(* Logix 5000 project; controller DispersionPlc vendor 1 type 14 code 108 rev 34.11; software revision 34.01; part 4 of 22 *)
(* tags used below, declared in another part *)
   _JISdebug : DINT;
   AFI : BOOL;
   B4320_HighHighLevel : BOOL;
   B4320_HighLevel : BOOL;
   B4320_OkToRun : BOOL;
   B4320_PumpAutoCommand : BOOL;
   B4320_Selected : BOOL;
   B4320_SelectPB : BOOL;
   B4320_Toggle : AOI_Toggle;
   B4320_Transfer : BOOL;
   B4320_transfer_amount : REAL;
   B4320_TransferLimit : REAL;
   B4320_transferLimitMessage : BOOL;
   B4320_TransferSetpoint : REAL;
   B4320_TransferStarted : BOOL;
   B4320_TransferStartPB : BOOL;
   B4320_TransferStopPB : BOOL;
   BL_4310_AUX : ALIAS FOR Local:1:I.Data[1].2;
   BL_4310_RUN : ALIAS FOR Local:1:O.Data[0].2;
   BLANK64 : Stp64;
   bogus_bit : BOOL;
   Cat_Pump_manual : BOOL;
   Cat_Recirc_Transfer_T430X : Seq64;
   Cat_Scale_Factor : REAL;
   cat_start_dispencse : BOOL;
   Cat_Tank_Destination : DINT;
   cat_target_weight_bypass : BOOL;
   Cat_Zero : REAL;
   catalyst_MaxFeedRate : REAL;
   CATALYST_RESET : BOOL;
   CatalystTimers_11_HMI : REAL;
   CE_4301 : REAL;
   CE_4301_OffSet : REAL;
   CE_4301_Sf : REAL;
   CurrentTrasferredLb : REAL;
   dan5 : BOOL;
   DATAFDUNLATCH : TIMER;
   DATAUNCOUNT : COUNTER;
   DispersionAlarms : BOOL[256];
   DPT_4301 : REAL;
   DPT_4301_Holding : REAL;
   DPT_4301_OffSet : REAL;
   DPT_4301_Samples : DINT;
   DPT_4301_Sf : REAL;
   DPT_4302 : REAL;
   DPT_4302_Holding : REAL;
   DPT_4302_OffSet : REAL;
   DPT_4302_Samples : DINT;
   DPT_4302_Sf : REAL;
   DPT_4303 : REAL;
   DPT_4303_Holding : REAL;
   DPT_4303_OffSet : REAL;
   DPT_4303_Samples : DINT;
   DPT_4303_Sf : REAL;
   DPT_4320 : REAL;
   Emergency_Cool_4301 : BOOL;
   Estop_Disp : ALIAS FOR Local:3:I.Data.1;
   Estop_Inx : ALIAS FOR Local:3:I.Data.3;
   FE_4303 : REAL;
   FE_4303_AOI : Analog_Scale;
   FE_4303_Corrected : REAL;
   FE_4303_Correction_Sf : REAL;
   FE_4303_OffSet : REAL;
   FE_4303_OffSet_Out : REAL;
   FE_4303_Out : REAL;
   FE_4304 : REAL;
   FE_4304_AOI : Analog_Scale;
   FE_4304_OffSet : REAL;
   FE_4304_Sf : REAL;
   FE_4305 : REAL;
   FE_4305_OffSet : REAL;
   FE_4305_Sf : REAL;
   INX_Alarm : BOOL[32];
   INX_AlarmTmr : TIMER[32];
   InxAlarms : BOOL[128];
   LS_4302_Raw : INT;
   MAINT_SV4304_02_PB : BOOL;
   MAINT_SV4304_03_PB : BOOL;
   MAINT_XV4304_04_PB : BOOL;
   MIXER_A_4304_RUN : ALIAS FOR Local:1:O.Data[0].16;
   MMI_A_4304_RUN_PB : BOOL;
   MMI_B4320_Level : INT;
   MMI_Cat_Nit_Purge_Time : REAL;
   MMI_Cat_Recirc_Pump_Speed : REAL;
   MMI_P_4304_RUN_PB : BOOL;
   MMI_P_4320_RUN_PB : BOOL;
   MMI_SV4304_02_PB : BOOL;
   MMI_SV4304_03_PB : BOOL;
   MMI_SV4304_PB : BOOL;
   MMI_T4301_Level : INT;
   MMI_T4302_Level : INT;
   MMI_V4304_Acc_Weight : REAL;
   MMI_V4304_Acc_Weight_Temp : REAL;
   MMI_V4304_TransTime_SP : REAL;
   MMI_V4304_Weight_SP : REAL;
   MMI_W4303_Level : INT;
   MMI_XV4304_02_PB : BOOL;
   MMI_XV4304_03_PB : BOOL;
   MMI_XV4304_04_PB : BOOL;
   MMI_XV_4304_01_PB : BOOL;
   O5_6_PL : ALIAS FOR Local:5:O.Data.14;
   O5_9_PL : ALIAS FOR Local:5:O.Data.9;
   O7_11_BEC : ALIAS FOR Local:7:O.Data.11;
   ONS101 : BOOL;
   PLCStatus : AStd_PLCStatus;
   S47_HighHighLevel : BOOL;
   S47_SelectPB : BOOL;
   S47_TransferStarted : BOOL;
   SPARE_O603 : ALIAS FOR Local:6:O.Data.3;
   SPARE_O604 : ALIAS FOR Local:6:O.Data.4;
   SRT_PB_BL_4310 : ALIAS FOR Local:2:I.Data.13;
   SRT_PB_P_4310 : ALIAS FOR Local:2:I.Data.15;
   STP_PB_BL_4310 : ALIAS FOR Local:2:I.Data.14;
   STP_PB_P_4310 : ALIAS FOR Local:3:I.Data.0;
   SV_4304 : ALIAS FOR Local:5:O.Data.11;
   SV_4304_02 : BOOL;
   SV_4304_02_Enable_PB : BOOL;
   SV_4304_03 : BOOL;
   SV_4304_03_Enable_PB : BOOL;
   SV_4310 : ALIAS FOR Local:5:O.Data.5;
   T4301_AIR_PURGE_AUTO : BOOL;
   T4301_AIR_PURGE_REQUEST : BOOL;
   T4301_COOLING_NOT_PURGED : BOOL;
   T4301_COOLING_OCCURED : BOOL;
   T4301_COOLING_OPERATION : BOOL;
   T4301_K : Kettle;
   T4301_Manual_AIR_PURGE_REQUEST : BOOL;
   T4301_Mixer : VFD;
   T4301_Post_PurgeTm : DINT;
   T4301_Pre_PurgeTm : DINT;
   T4301_Process_Alarm_Setpoints : Alarm_SPT;
   T4301_Purge_Complete : BOOL;
   T4301_Request_Cooling_Tmr : TIMER[5];
   T4301Purge : Seq64;
   T_4301_Temp_Holding : REAL;
   T_4301_Temp_Samples : REAL;
   Task_Permissive : DINT[2];
   TE_4301A : ALIAS FOR Local:8:I.Ch0Data;
   TOGGLE : BOOL;
   TransferDone : BOOL;
   TransferSetpoint : REAL;
   V4304_Pump : VFD;
   V4304_Pump_TargetDriveSpeed_Timer : TIMER;
   XV_4304 : ALIAS FOR Local:5:O.Data.4;
   XV_4304_02 : BOOL;
   XV_4304_03 : BOOL;
   XV_4304_04 : BOOL;
   XV_S47_1_CloseCommand : BOOL;
   XV_S47_1_IsClosed : BOOL;
   XV_S47_1_IsOpen : BOOL;
   XV_S47_1_OpenCommand : BOOL;
   XV_S47_2_CloseCommand : BOOL;
   XV_S47_2_IsClosed : BOOL;
   ZSO_4304_02 : BOOL;
   ZSO_4304_03 : BOOL;
(* General_Purpose, continued *)

ROUTINE TimeSync   (* ladder *)
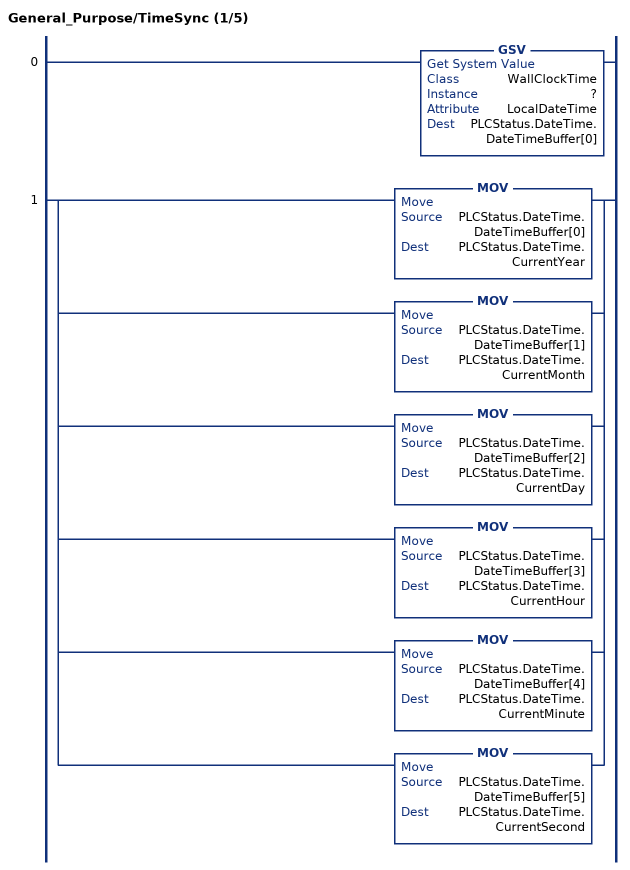
   0: GSV(WallClockTime,?,LocalDateTime,PLCStatus.DateTime.DateTimeBuffer[0]);
   1: [MOV(PLCStatus.DateTime.DateTimeBuffer[0],PLCStatus.DateTime.CurrentYear) ,MOV(PLCStatus.DateTime.DateTimeBuffer[1],PLCStatus.DateTime.CurrentMonth) ,MOV(PLCStatus.DateTime.DateTimeBuffer[2],PLCStatus.DateTime.CurrentDay) ,MOV(PLCStatus.DateTime.DateTimeBuffer[3],PLCStatus.DateTime.CurrentHour) ,MOV(PLCStatus.DateTime.DateTimeBuffer[4],PLCStatus.DateTime.CurrentMinute) ,MOV(PLCStatus.DateTime.DateTimeBuffer[5],PLCStatus.DateTime.CurrentSecond) ];
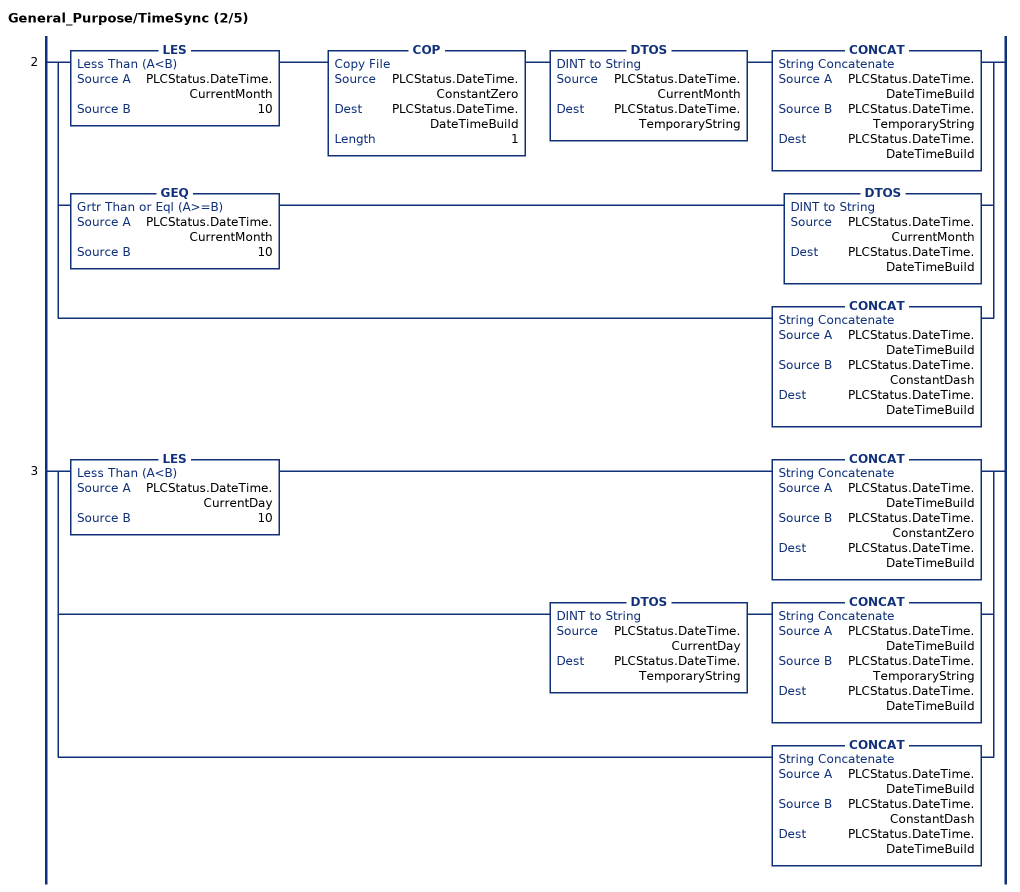
   2: [LES(PLCStatus.DateTime.CurrentMonth,10) COP(PLCStatus.DateTime.ConstantZero,PLCStatus.DateTime.DateTimeBuild,1) DTOS(PLCStatus.DateTime.CurrentMonth,PLCStatus.DateTime.TemporaryString) CONCAT(PLCStatus.DateTime.DateTimeBuild,PLCStatus.DateTime.TemporaryString,PLCStatus.DateTime.DateTimeBuild) ,GEQ(PLCStatus.DateTime.CurrentMonth,10) DTOS(PLCStatus.DateTime.CurrentMonth,PLCStatus.DateTime.DateTimeBuild) ,CONCAT(PLCStatus.DateTime.DateTimeBuild,PLCStatus.DateTime.ConstantDash,PLCStatus.DateTime.DateTimeBuild) ];
   3: [LES(PLCStatus.DateTime.CurrentDay,10) CONCAT(PLCStatus.DateTime.DateTimeBuild,PLCStatus.DateTime.ConstantZero,PLCStatus.DateTime.DateTimeBuild) ,DTOS(PLCStatus.DateTime.CurrentDay,PLCStatus.DateTime.TemporaryString) CONCAT(PLCStatus.DateTime.DateTimeBuild,PLCStatus.DateTime.TemporaryString,PLCStatus.DateTime.DateTimeBuild) ,CONCAT(PLCStatus.DateTime.DateTimeBuild,PLCStatus.DateTime.ConstantDash,PLCStatus.DateTime.DateTimeBuild) ];
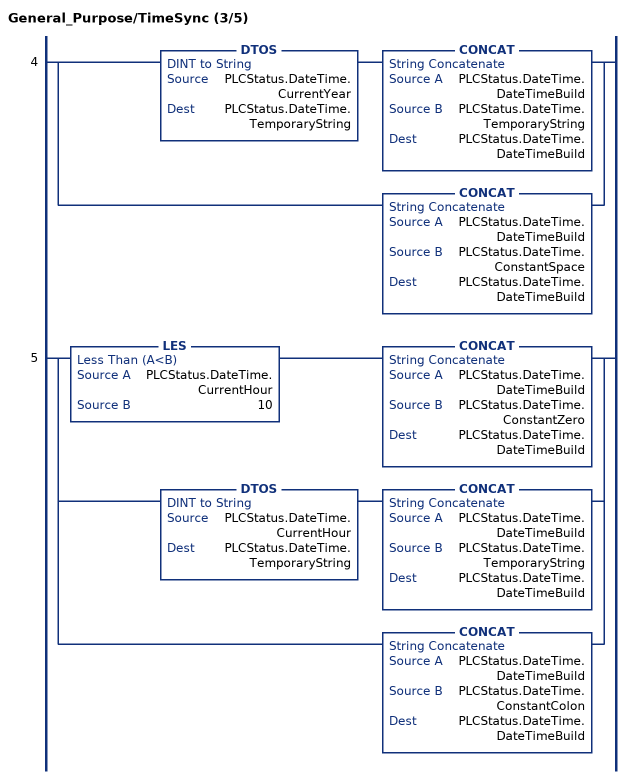
   4: [DTOS(PLCStatus.DateTime.CurrentYear,PLCStatus.DateTime.TemporaryString) CONCAT(PLCStatus.DateTime.DateTimeBuild,PLCStatus.DateTime.TemporaryString,PLCStatus.DateTime.DateTimeBuild) ,CONCAT(PLCStatus.DateTime.DateTimeBuild,PLCStatus.DateTime.ConstantSpace,PLCStatus.DateTime.DateTimeBuild) ];
   5: [LES(PLCStatus.DateTime.CurrentHour,10) CONCAT(PLCStatus.DateTime.DateTimeBuild,PLCStatus.DateTime.ConstantZero,PLCStatus.DateTime.DateTimeBuild) ,DTOS(PLCStatus.DateTime.CurrentHour,PLCStatus.DateTime.TemporaryString) CONCAT(PLCStatus.DateTime.DateTimeBuild,PLCStatus.DateTime.TemporaryString,PLCStatus.DateTime.DateTimeBuild) ,CONCAT(PLCStatus.DateTime.DateTimeBuild,PLCStatus.DateTime.ConstantColon,PLCStatus.DateTime.DateTimeBuild) ];
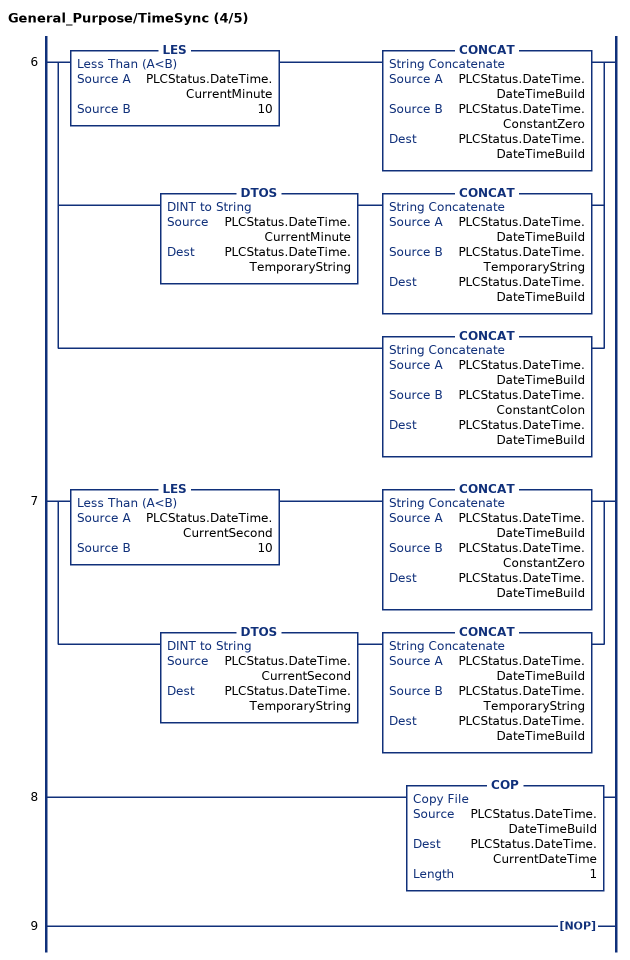
   6: [LES(PLCStatus.DateTime.CurrentMinute,10) CONCAT(PLCStatus.DateTime.DateTimeBuild,PLCStatus.DateTime.ConstantZero,PLCStatus.DateTime.DateTimeBuild) ,DTOS(PLCStatus.DateTime.CurrentMinute,PLCStatus.DateTime.TemporaryString) CONCAT(PLCStatus.DateTime.DateTimeBuild,PLCStatus.DateTime.TemporaryString,PLCStatus.DateTime.DateTimeBuild) ,CONCAT(PLCStatus.DateTime.DateTimeBuild,PLCStatus.DateTime.ConstantColon,PLCStatus.DateTime.DateTimeBuild) ];
   7: [LES(PLCStatus.DateTime.CurrentSecond,10) CONCAT(PLCStatus.DateTime.DateTimeBuild,PLCStatus.DateTime.ConstantZero,PLCStatus.DateTime.DateTimeBuild) ,DTOS(PLCStatus.DateTime.CurrentSecond,PLCStatus.DateTime.TemporaryString) CONCAT(PLCStatus.DateTime.DateTimeBuild,PLCStatus.DateTime.TemporaryString,PLCStatus.DateTime.DateTimeBuild) ];
   8: COP(PLCStatus.DateTime.DateTimeBuild,PLCStatus.DateTime.CurrentDateTime,1);
   9: NOP();
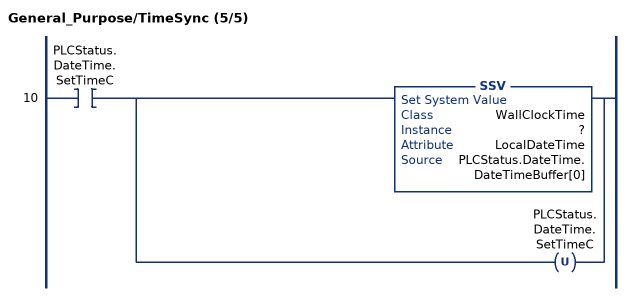
   10: XIC(PLCStatus.DateTime.SetTimeC)[SSV(WallClockTime,?,LocalDateTime,PLCStatus.DateTime.DateTimeBuffer[0]) ,OTU(PLCStatus.DateTime.SetTimeC) ];
END_ROUTINE
END_PROGRAM

PROGRAM MainProgram   (* main routine MainRoutine *)
VAR
   AllwaysOff : BOOL;
   B4320_Tank_Max_Lbs : REAL := 50817.0;
   BarcodeBypassAcitve1 : BOOL;
   BarcodeBypassAcitvePB1 : BOOL;
   BebugBit : BOOL[32] := ([0] := 1, [1] := 1, [2] := 1, [3] := 1, [4] := 1, [5] := 1, [6] := 1, [7] := 1, [8] := 1, [9] := 1, [10] := 1, [11] := 1, [12] := 1, [13] := 1, [14] := 1, [15] := 1, [16] := 1);
   block : BOOL;
   BypassOns : BOOL;
   calculated_percent : DINT := 50;
   Catalyst_FlowTimer : TIMER := (PRE := 1000, ACC := 84, EN := 1, TT := 1);
   Catalyst_OneShots : BOOL[32];
   catalyst_Target_Wgt_Lb_Min : REAL := 1.575;
   Catalyst_Timers : TIMER[20] := ([0].PRE := 20000, [11].PRE := 7000);
   CatDispenced_Snapshot : REAL := 0.027864583;
   Check4AsciiLine : SERIAL_PORT_CONTROL := (EU := 1, DN := 1, EM := 1);
   D_Alarm_11_Timer : TIMER := (PRE := 1000);
   D_Alarm_9_Timer : TIMER := (PRE := 1000);
   D_AlarmTimers : TIMER[200] := ([0].PRE := 3000, [13].PRE := 2000, [14].PRE := 3000, [15].PRE := 3000, [18].PRE := 3000, [24].PRE := 3000, [27].PRE := 3000, [28].PRE := 3000, [38].PRE := 5000, [44].PRE := 3000, [45].PRE := 4000, [50].PRE := 3000, [52].PRE := 3000, [54].PRE := 3000, [55].PRE := 60000, [65].PRE := 2000, [68].PRE := 10000, [70].PRE := 3000, [71].PRE := 5000, [74].PRE := 3000, [77].PRE := 3000, [87].PRE := 2000, [88].PRE := 2000, [89].PRE := 5000, [90].PRE := 5000, [91].PRE := 5000, [92].PRE := 5000, [93].PRE := 5000, [94].PRE := 5000, [95].PRE := 5000, [96].PRE := 3000, [97].PRE := 1000, [98].PRE := 1000, [99].PRE := 1000, [101].PRE := 3000, [102].PRE := 3000, [103].PRE := 3000, [104].PRE := 3000, [105].PRE := 3000, [106].PRE := 3000, [144].PRE := 3000, [145].PRE := 3000, [146].PRE := 3000, [147].PRE := 3000, [148].PRE := 3000, [149].PRE := 3000, [150].PRE := 1000, [151].PRE := 1000, [152].PRE := 3000);
   D_AlarmTimers2 : TIMER[100] := ([0].PRE := 1000, [1].PRE := 1000, [2].PRE := 5000, [3].PRE := 5000, [3].ACC := 5009, [3].EN := 1, [3].DN := 1, [11].PRE := 2000, [12].PRE := 2000, [13].PRE := 2000, [14].PRE := 2000, [15].PRE := 2000, [16].PRE := 2000, [17].PRE := 2000, [18].PRE := 2000, [19].PRE := 20000, [20].PRE := 2000, [21].PRE := 5000, [22].PRE := 5000);
   DataBufferRead : SERIAL_PORT_CONTROL := (LEN := 82, POS := 13, EU := 1, EM := 1);
   DataFromBuffer : STRING := '$02     843LN $0D';
   Disp_AlarmScanIdx : DINT := 103;
   Disp_NewAlarmScanIdx : DINT := 112;
   Disp_Ons : BOOL[32];
   DispAlarmDisplayTmr : TIMER := (PRE := 3500, ACC := 2813, EN := 1, TT := 1);
   DispersionAckAlarms : BOOL[128] := ([2] := 1, [103] := 1, [108] := 1);
   DispersionProductID_BarcodeScan : STRING := '813143575381';
   DispersionProductID_ScanIndex_Storage : DINT := 2;
   DispersionProductIDEntryStorage : STRING := '8132028';
   DispersionProductIDMatch : DINT := 1;
   Dispertion_Intelock_Status : BOOL := 1;
   Dn_DataMap_In : INT[12] := ([0] := 3597);
   Dn_DataMap_out : INT[12] := ([1] := 4530);
   DnEnable : BOOL := 1;
   DPT_4303_Warn : REAL := 15500.0;
   DPT_4304_Tare_Val : REAL;
   DPT_4320_Holding : REAL := 14396.196;
   DPT_4320_Samples : DINT := 100;
   Fcv_4305_Temp : REAL;
   FCV_Rate : REAL := 5.0;
   FE_4303_Deaband_Minus : REAL := 1.0;
   FE_4303_Deaband_Plus : REAL := -1.0;
   FE_4303_Feed_Error : REAL := 0.23413277;
   FE_4303_Prop_Gain : REAL;
   FE_4303_Temp : REAL := 85.79976;
   FE_4304_Deaband_Minus : REAL := 0.07;
   FE_4304_Deaband_Plus : REAL := -0.07;
   FE_4304_Feed_Error : REAL := -0.084375024;
   FE_4304_Prop_Gain : REAL;
   FE_4304_Temp : REAL := 63.49997;
   FE_4305_Deaband_Minus : REAL := -0.8;
   FE_4305_Deaband_Plus : REAL := 0.8;
   FE_4305_Feed_Error : REAL := -142.616;
   gotcha : BOOL;
   InputIdx : DINT := 37;
   IntAlrTmr : TIMER[32] := ([0].PRE := 3000, [1].PRE := 3000, [2].PRE := 3000, [3].PRE := 10000, [6].PRE := 10000, [7].PRE := 10000, [14].PRE := 2000, [15].PRE := 1000, [16].PRE := 1000, [17].PRE := 1000, [18].PRE := 1000, [19].PRE := 1000, [22].PRE := 1000);
   Inx_AlarmsResetting : BOOL;
   Inx_AlrResetIdx : DINT := 127;
   Inx_NewAlarmScanIdx : DINT := 10;
   inx_QuedAlarm : DINT := 11;
   InxAckAlarms : BOOL[128] := ([11] := 1);
   InxAlarmDisplayTmr : TIMER := (PRE := 3500, ACC := 1255, EN := 1, TT := 1);
   InxTog : BOOL[32];
   Messaging_Timer2 : TIMER := (PRE := 750, EN := 1, TT := 1);
   MMI_RO_Acc_weight : REAL := 200.37845;
   MMI_SV4303_01_PB : BOOL;
   MMI_V4303_Acc_weight : REAL := 3245941.2;
   MMI_v4304_Acc_Weight_Reset : BOOL;
   MonDispenced_Snapshot : REAL := 0.3650133;
   Monomer_FlowTimer : TIMER := (PRE := 1000, ACC := 1004, EN := 1, DN := 1);
   Monomer_OneShots : BOOL[32];
   Monomer_Target_Wgt_Lb_Min : REAL := 21.666666;
   MonomerTimers : TIMER[12] := ([0].PRE := 10000);
   New_InxAlarmDetected : BOOL;
   No_Disp_Alarms : BOOL;
   No_Inx_Alarms : BOOL;
   NoNEwAlarmsDestedted : BOOL := 1;
   NoNEwInxAlarmsDestedted : BOOL := 1;
   ONS : BOOL[32] := ([2] := 1);
   ons100 : BOOL := 1;
   OutPutIdx : DINT := 17;
   P4303_Rate : REAL := 0.2;
   P4304_Rate : REAL := 0.3;
   ReffBit : BOOL;
   Ro_FlowTimer : TIMER := (PRE := 1000);
   Ro_Ons : BOOL[32];
   Ro_RampTimer : TIMER := (PRE := 500);
   Ro_Target_Wgt_Lb_Min : REAL := 100.0;
   RoDispenced_Snapshot : REAL := 1.5442973;
   ScnCnt : DINT;
   SV_4303_03_Man_Override : BOOL;
   T4301_T4302_Xfer_In_Enable : BOOL := 1;
   T4301_Tank_Max_Lbs : REAL := 56500.0;
   T4301Ons : BOOL[32] := ([11] := 1, [14] := 1, [19] := 1, [20] := 1, [21] := 1, [27] := 1, [28] := 1, [29] := 1, [31] := 1);
   T4302_Tank_Max_Lbs : REAL := 56500.0;
   T4302Ons : BOOL[32] := ([11] := 1, [14] := 1, [21] := 1, [27] := 1, [28] := 1, [29] := 1, [31] := 1);
   Temp : BOOL := 1;
   TempRoValveVal : INT := 4640;
   TEST_BIT : BOOL;
   TestBit : AB:1769_DI16:I:0;
   TestBitt : BOOL := 1;
   TestDispValves : BOOL := 1;
   TestTog : BOOL;
   TmpInxAlr : BOOL;
   TogResult : BOOL;
   TurningOnReffBit : BOOL;
   V4304_RampTimer : TIMER := (PRE := 1000, ACC := 84, EN := 1, TT := 1);
   VfdReff : VFD := (TargetDriveSpeed := 30, I_Ready := 1, I_CmdDir := 1, I_ActDir := 1, I_LocalContStat1 := 1, I_LocalContStat2 := 1, I_LocalContStat3 := 1, O_V_CmdReff := 4530.0, SpeedScaleIn := 151.0, SpeedScaleOut := 151.0, MaxOutPut := 100.0, MinOutput := 10.0);
   W4303_RampTimer : TIMER := (PRE := 500, ACC := 340, EN := 1, TT := 1);
   W4303_Tank_Max_Lbs : REAL := 16400.0;
   ZS_4301_timer : TIMER := (PRE := 3000, ACC := 3010, EN := 1, DN := 1);
   ZS_4302_timer : TIMER := (PRE := 3000);
END_VAR

ROUTINE AirPurge   (* ladder *)
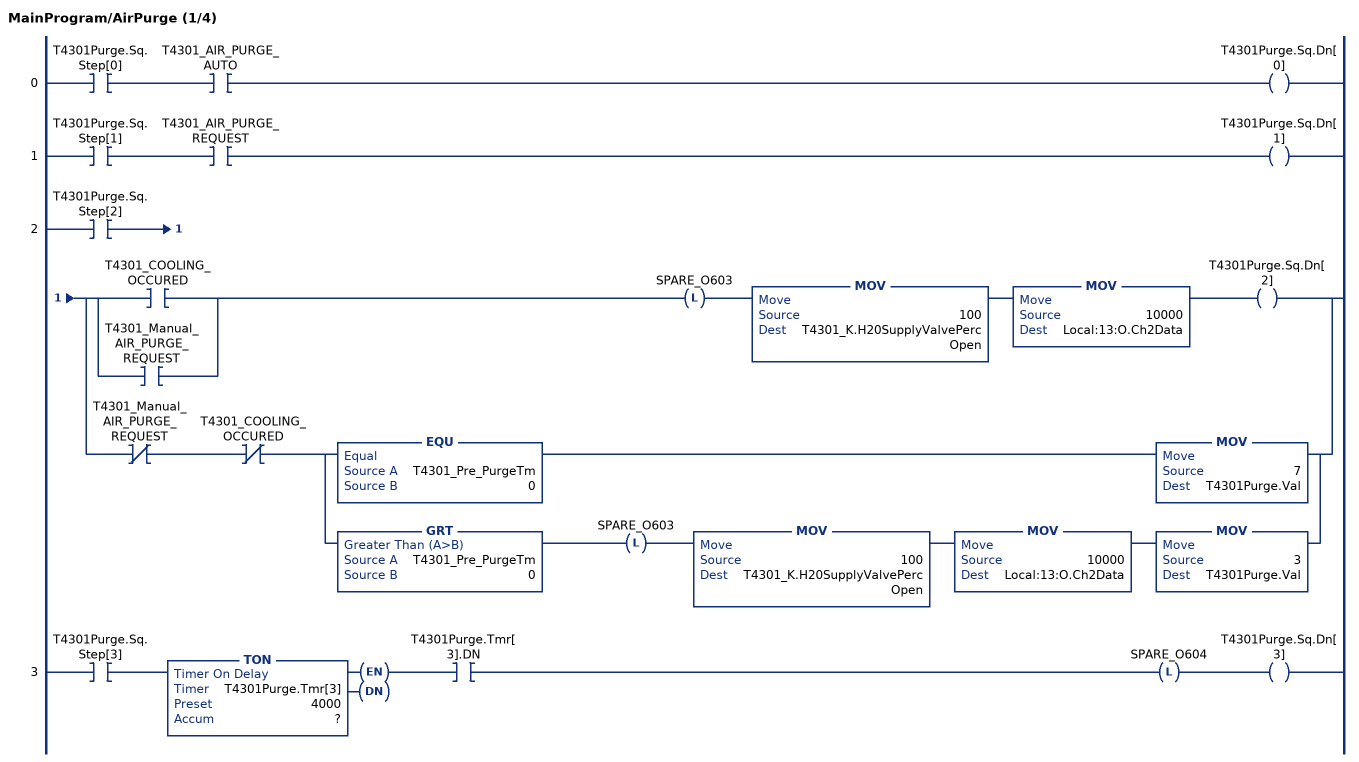
   0: XIC(T4301Purge.Sq.Step[0])XIC(T4301_AIR_PURGE_AUTO)OTE(T4301Purge.Sq.Dn[0]);
   1: XIC(T4301Purge.Sq.Step[1])XIC(T4301_AIR_PURGE_REQUEST)OTE(T4301Purge.Sq.Dn[1]);
   2: XIC(T4301Purge.Sq.Step[2])[[XIC(T4301_COOLING_OCCURED) ,XIC(T4301_Manual_AIR_PURGE_REQUEST) ] OTL(SPARE_O603) MOV(100,T4301_K.H20SupplyValvePercOpen) MOV(10000,Local:13:O.Ch2Data) OTE(T4301Purge.Sq.Dn[2]) ,XIO(T4301_Manual_AIR_PURGE_REQUEST) XIO(T4301_COOLING_OCCURED) [EQU(T4301_Pre_PurgeTm,0) MOV(7,T4301Purge.Val) ,GRT(T4301_Pre_PurgeTm,0) OTL(SPARE_O603) MOV(100,T4301_K.H20SupplyValvePercOpen) MOV(10000,Local:13:O.Ch2Data) MOV(3,T4301Purge.Val) ] ];
   3: XIC(T4301Purge.Sq.Step[3])TON(T4301Purge.Tmr[3],?,?)XIC(T4301Purge.Tmr[3].DN)OTL(SPARE_O604)OTE(T4301Purge.Sq.Dn[3]);
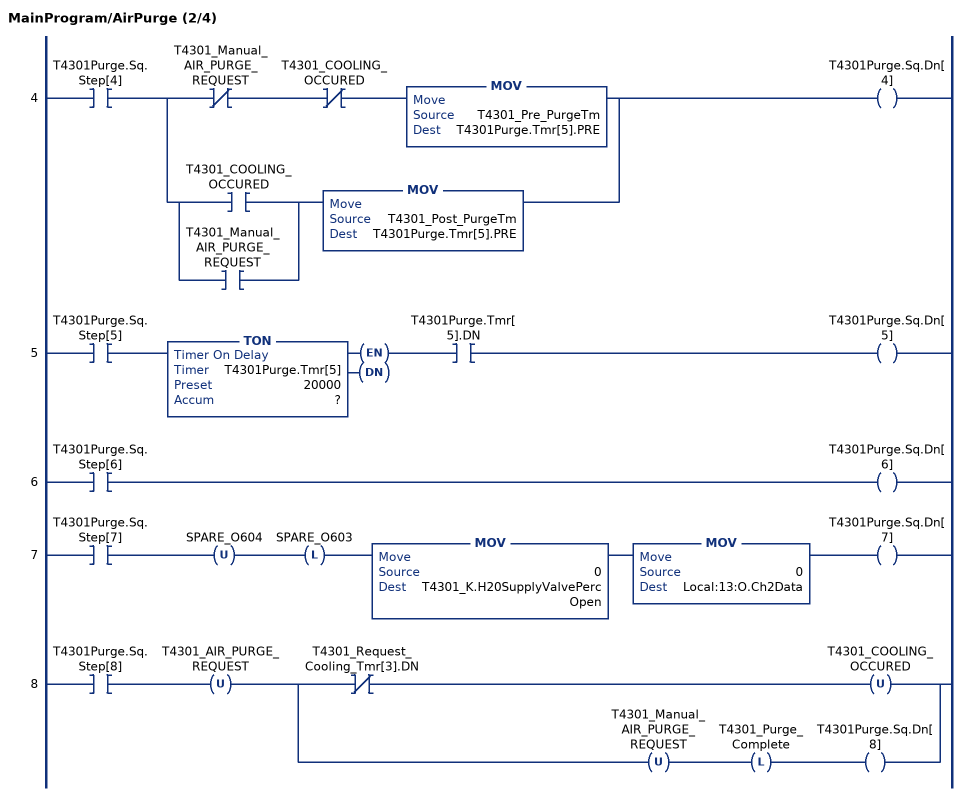
   4: XIC(T4301Purge.Sq.Step[4])[XIO(T4301_Manual_AIR_PURGE_REQUEST) XIO(T4301_COOLING_OCCURED) MOV(T4301_Pre_PurgeTm,T4301Purge.Tmr[5].PRE) ,[XIC(T4301_COOLING_OCCURED) ,XIC(T4301_Manual_AIR_PURGE_REQUEST) ] MOV(T4301_Post_PurgeTm,T4301Purge.Tmr[5].PRE) ]OTE(T4301Purge.Sq.Dn[4]);
   5: XIC(T4301Purge.Sq.Step[5])TON(T4301Purge.Tmr[5],?,?)XIC(T4301Purge.Tmr[5].DN)OTE(T4301Purge.Sq.Dn[5]);
   6: XIC(T4301Purge.Sq.Step[6])OTE(T4301Purge.Sq.Dn[6]);
   7: XIC(T4301Purge.Sq.Step[7])OTU(SPARE_O604)OTL(SPARE_O603)MOV(0,T4301_K.H20SupplyValvePercOpen)MOV(0,Local:13:O.Ch2Data)OTE(T4301Purge.Sq.Dn[7]);
   8: XIC(T4301Purge.Sq.Step[8])OTU(T4301_AIR_PURGE_REQUEST)[XIO(T4301_Request_Cooling_Tmr[3].DN) OTU(T4301_COOLING_OCCURED) ,OTU(T4301_Manual_AIR_PURGE_REQUEST) OTL(T4301_Purge_Complete) OTE(T4301Purge.Sq.Dn[8]) ];
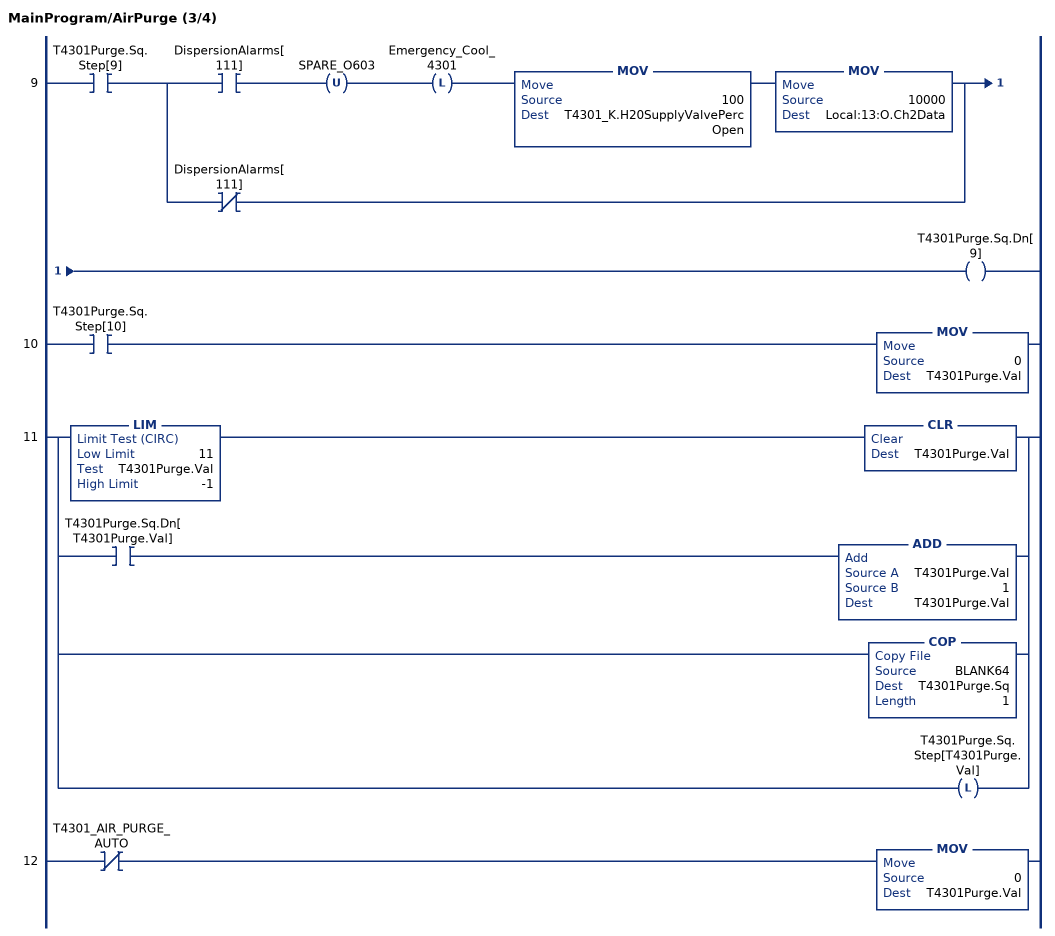
   9: XIC(T4301Purge.Sq.Step[9])[XIC(DispersionAlarms[111]) OTU(SPARE_O603) OTL(Emergency_Cool_4301) MOV(100,T4301_K.H20SupplyValvePercOpen) MOV(10000,Local:13:O.Ch2Data) ,XIO(DispersionAlarms[111]) ]OTE(T4301Purge.Sq.Dn[9]);
   10: XIC(T4301Purge.Sq.Step[10])MOV(0,T4301Purge.Val);
   11: [LIM(11,T4301Purge.Val,-1) CLR(T4301Purge.Val) ,XIC(T4301Purge.Sq.Dn[T4301Purge.Val]) ADD(T4301Purge.Val,1,T4301Purge.Val) ,COP(BLANK64,T4301Purge.Sq,1) ,OTL(T4301Purge.Sq.Step[T4301Purge.Val]) ];
   12: XIO(T4301_AIR_PURGE_AUTO)MOV(0,T4301Purge.Val);
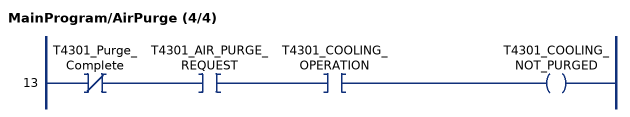
   13: XIO(T4301_Purge_Complete)XIC(T4301_AIR_PURGE_REQUEST)XIC(T4301_COOLING_OPERATION)OTE(T4301_COOLING_NOT_PURGED);
END_ROUTINE

ROUTINE Ammonium_Hyd   (* ladder *)
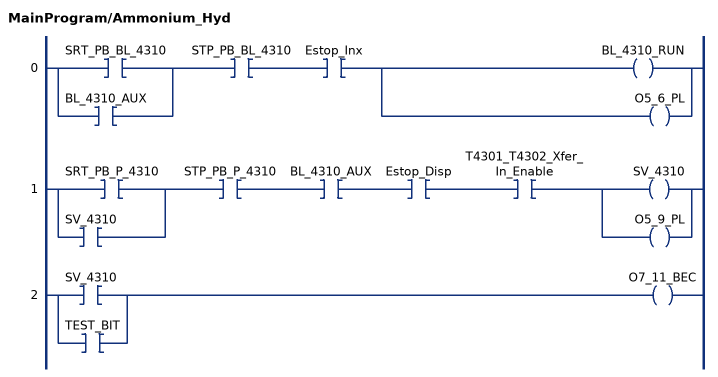
   0: [XIC(SRT_PB_BL_4310) ,XIC(BL_4310_AUX) ]XIC(STP_PB_BL_4310)XIC(Estop_Inx)[OTE(BL_4310_RUN) ,OTE(O5_6_PL) ];
   1: [XIC(SRT_PB_P_4310) ,XIC(SV_4310) ]XIC(STP_PB_P_4310)XIC(BL_4310_AUX)XIC(Estop_Disp)XIC(T4301_T4302_Xfer_In_Enable)[OTE(SV_4310) ,OTE(O5_9_PL) ];
   2: [XIC(SV_4310) ,XIC(TEST_BIT) ]OTE(O7_11_BEC);
END_ROUTINE

ROUTINE ANALOGS   (* ladder *)
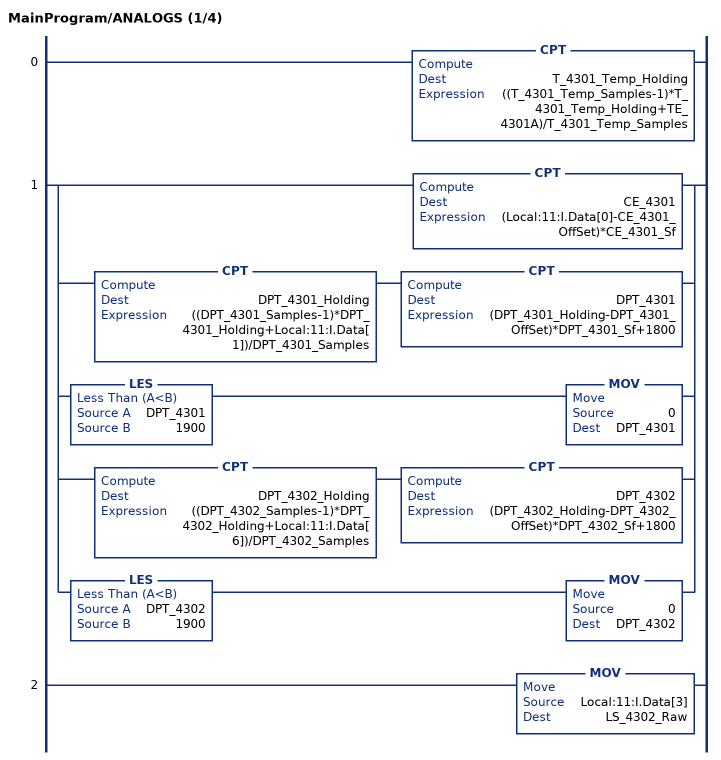
   0: CPT(T_4301_Temp_Holding,((T_4301_Temp_Samples-1)*T_4301_Temp_Holding+TE_4301A)/T_4301_Temp_Samples);
   1: [CPT(CE_4301,(Local:11:I.Data[0]-CE_4301_OffSet)*CE_4301_Sf) ,CPT(DPT_4301_Holding,((DPT_4301_Samples-1)*DPT_4301_Holding+Local:11:I.Data[1])/DPT_4301_Samples) CPT(DPT_4301,(DPT_4301_Holding-DPT_4301_OffSet)*DPT_4301_Sf+1800) ,LES(DPT_4301,1900) MOV(0,DPT_4301) ,CPT(DPT_4302_Holding,((DPT_4302_Samples-1)*DPT_4302_Holding+Local:11:I.Data[6])/DPT_4302_Samples) CPT(DPT_4302,(DPT_4302_Holding-DPT_4302_OffSet)*DPT_4302_Sf+1800) ,LES(DPT_4302,1900) MOV(0,DPT_4302) ];
   2: MOV(Local:11:I.Data[3],LS_4302_Raw);
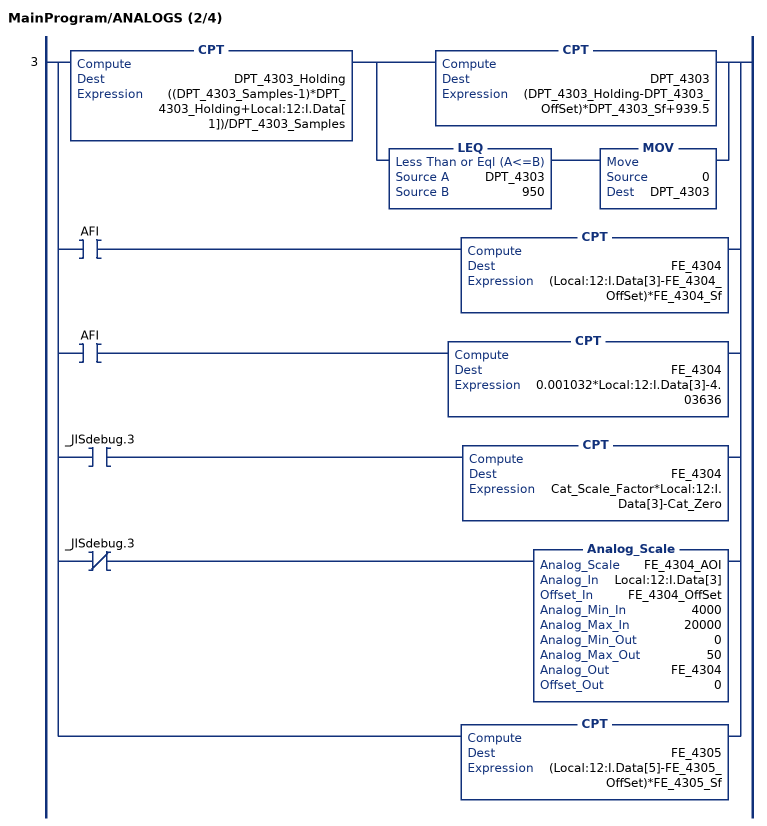
   3: [CPT(DPT_4303_Holding,((DPT_4303_Samples-1)*DPT_4303_Holding+Local:12:I.Data[1])/DPT_4303_Samples) [CPT(DPT_4303,(DPT_4303_Holding-DPT_4303_OffSet)*DPT_4303_Sf+939.5) ,LEQ(DPT_4303,950) MOV(0,DPT_4303) ] ,[XIC(AFI) CPT(FE_4304,(Local:12:I.Data[3]-FE_4304_OffSet)*FE_4304_Sf) ,XIC(AFI) CPT(FE_4304,0.001032*Local:12:I.Data[3]-4.03636) ,XIC(_JISdebug.3) CPT(FE_4304,Cat_Scale_Factor*Local:12:I.Data[3]-Cat_Zero) ,XIO(_JISdebug.3) Analog_Scale(FE_4304_AOI,Local:12:I.Data[3],FE_4304_OffSet,4000,20000,0,50,FE_4304,0) ] ,CPT(FE_4305,(Local:12:I.Data[5]-FE_4305_OffSet)*FE_4305_Sf) ];
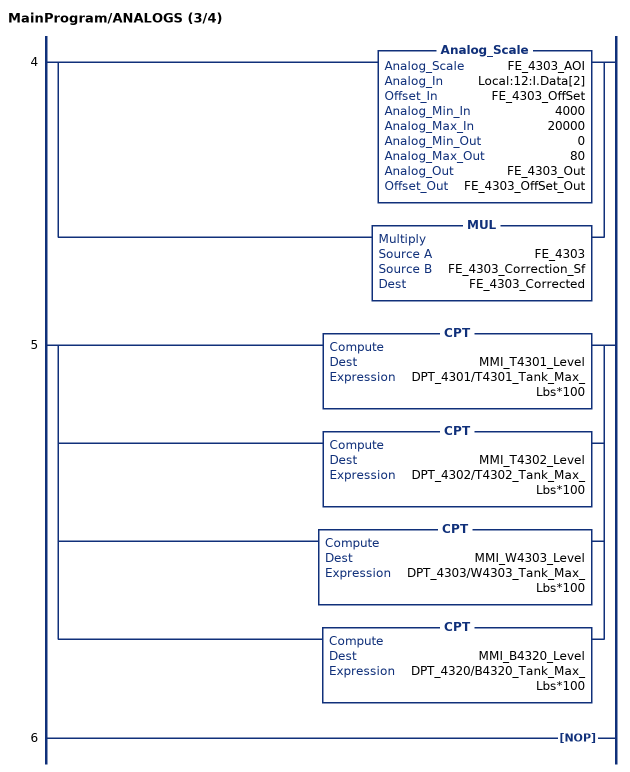
   4: [Analog_Scale(FE_4303_AOI,Local:12:I.Data[2],FE_4303_OffSet,4000,20000,0,80,FE_4303_Out,FE_4303_OffSet_Out) ,MUL(FE_4303,FE_4303_Correction_Sf,FE_4303_Corrected) ];
   5: [CPT(MMI_T4301_Level,DPT_4301/T4301_Tank_Max_Lbs*100) ,CPT(MMI_T4302_Level,DPT_4302/T4302_Tank_Max_Lbs*100) ,CPT(MMI_W4303_Level,DPT_4303/W4303_Tank_Max_Lbs*100) ,CPT(MMI_B4320_Level,DPT_4320/B4320_Tank_Max_Lbs*100) ];
   6: NOP();
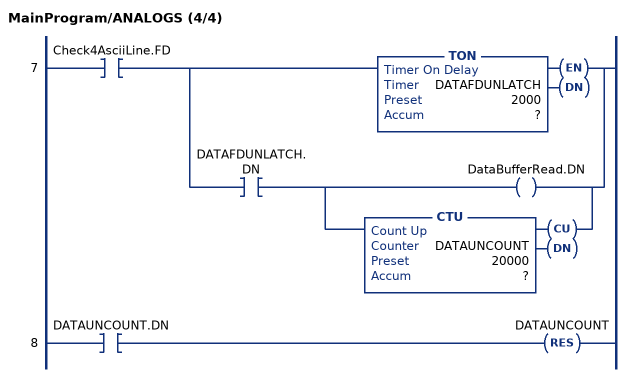
   7: XIC(Check4AsciiLine.FD)[TON(DATAFDUNLATCH,?,?) ,XIC(DATAFDUNLATCH.DN) [OTE(DataBufferRead.DN) ,CTU(DATAUNCOUNT,?,?) ] ];
   8: XIC(DATAUNCOUNT.DN)RES(DATAUNCOUNT);
END_ROUTINE

ROUTINE B4320_Transfer   (* ladder *)
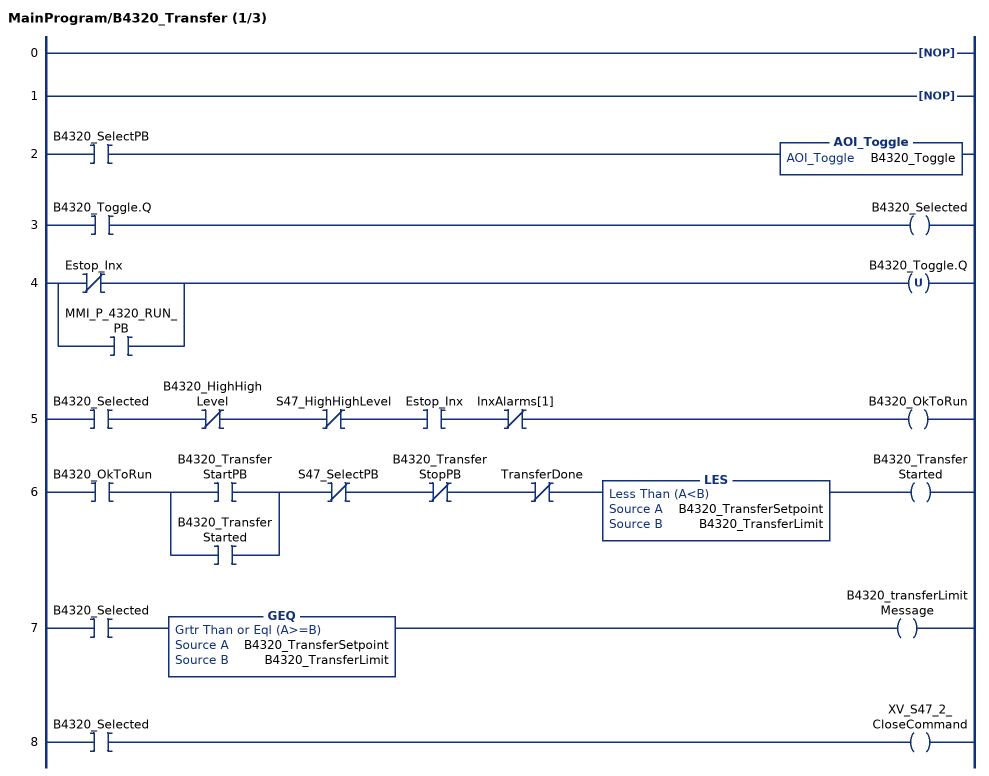
   0: NOP();
   1: NOP();
   2: XIC(B4320_SelectPB)AOI_Toggle(B4320_Toggle);
   3: XIC(B4320_Toggle.Q)OTE(B4320_Selected);
   4: [XIO(Estop_Inx) ,XIC(MMI_P_4320_RUN_PB) ]OTU(B4320_Toggle.Q);
   5: XIC(B4320_Selected)XIO(B4320_HighHighLevel)XIO(S47_HighHighLevel)XIC(Estop_Inx)XIO(InxAlarms[1])OTE(B4320_OkToRun);
   6: XIC(B4320_OkToRun)[XIC(B4320_TransferStartPB) ,XIC(B4320_TransferStarted) ]XIO(S47_SelectPB)XIO(B4320_TransferStopPB)XIO(TransferDone)LES(B4320_TransferSetpoint,B4320_TransferLimit)OTE(B4320_TransferStarted);
   7: XIC(B4320_Selected)GEQ(B4320_TransferSetpoint,B4320_TransferLimit)OTE(B4320_transferLimitMessage);
   8: XIC(B4320_Selected)OTE(XV_S47_2_CloseCommand);
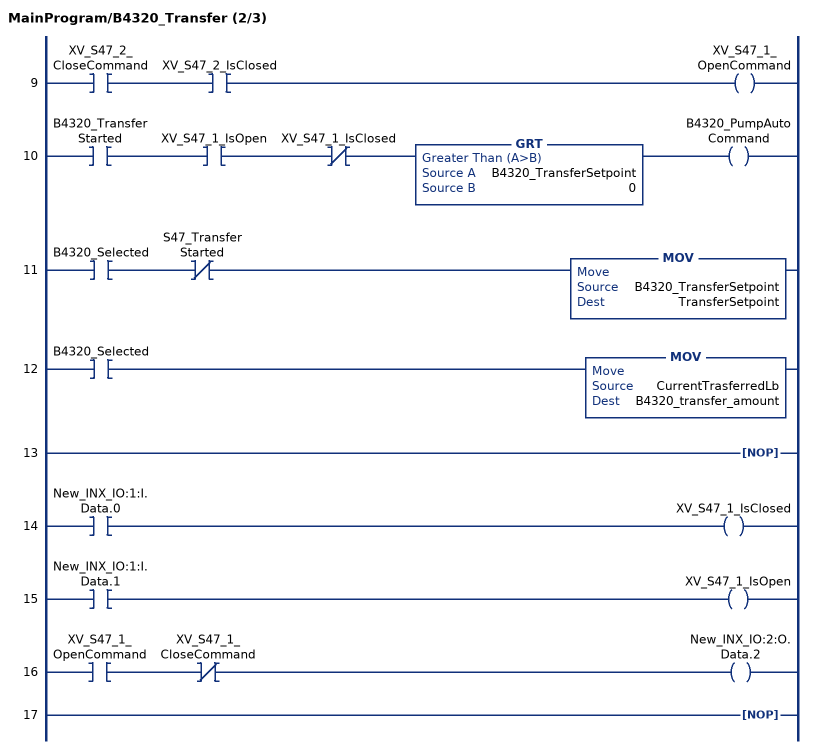
   9: XIC(XV_S47_2_CloseCommand)XIC(XV_S47_2_IsClosed)OTE(XV_S47_1_OpenCommand);
   10: XIC(B4320_TransferStarted)XIC(XV_S47_1_IsOpen)XIO(XV_S47_1_IsClosed)GRT(B4320_TransferSetpoint,0)OTE(B4320_PumpAutoCommand);
   11: XIC(B4320_Selected)XIO(S47_TransferStarted)MOV(B4320_TransferSetpoint,TransferSetpoint);
   12: XIC(B4320_Selected)MOV(CurrentTrasferredLb,B4320_transfer_amount);
   13: NOP();
   14: XIC(New_INX_IO:1:I.Data.0)OTE(XV_S47_1_IsClosed);
   15: XIC(New_INX_IO:1:I.Data.1)OTE(XV_S47_1_IsOpen);
   16: XIC(XV_S47_1_OpenCommand)XIO(XV_S47_1_CloseCommand)OTE(New_INX_IO:2:O.Data.2);
   17: NOP();
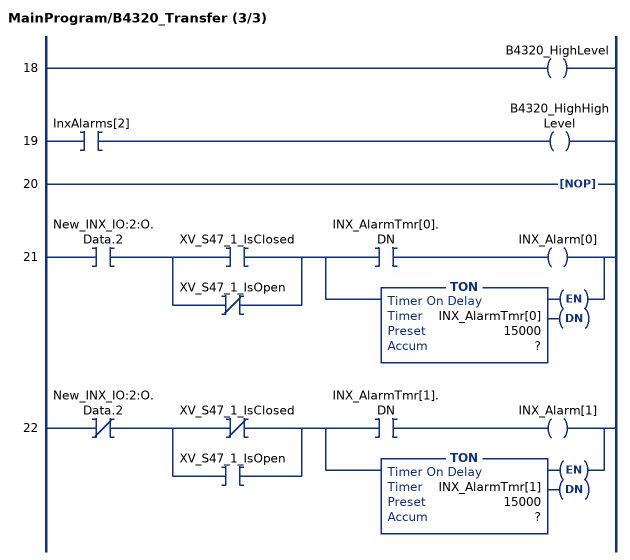
   18: OTE(B4320_HighLevel);
   19: XIC(InxAlarms[2])OTE(B4320_HighHighLevel);
   20: NOP();
   21: XIC(New_INX_IO:2:O.Data.2)[XIC(XV_S47_1_IsClosed) ,XIO(XV_S47_1_IsOpen) ][XIC(INX_AlarmTmr[0].DN) OTE(INX_Alarm[0]) ,TON(INX_AlarmTmr[0],?,?) ];
   22: XIO(New_INX_IO:2:O.Data.2)[XIO(XV_S47_1_IsClosed) ,XIC(XV_S47_1_IsOpen) ][XIC(INX_AlarmTmr[1].DN) OTE(INX_Alarm[1]) ,TON(INX_AlarmTmr[1],?,?) ];
END_ROUTINE

ROUTINE Catalyst   (* ladder *)
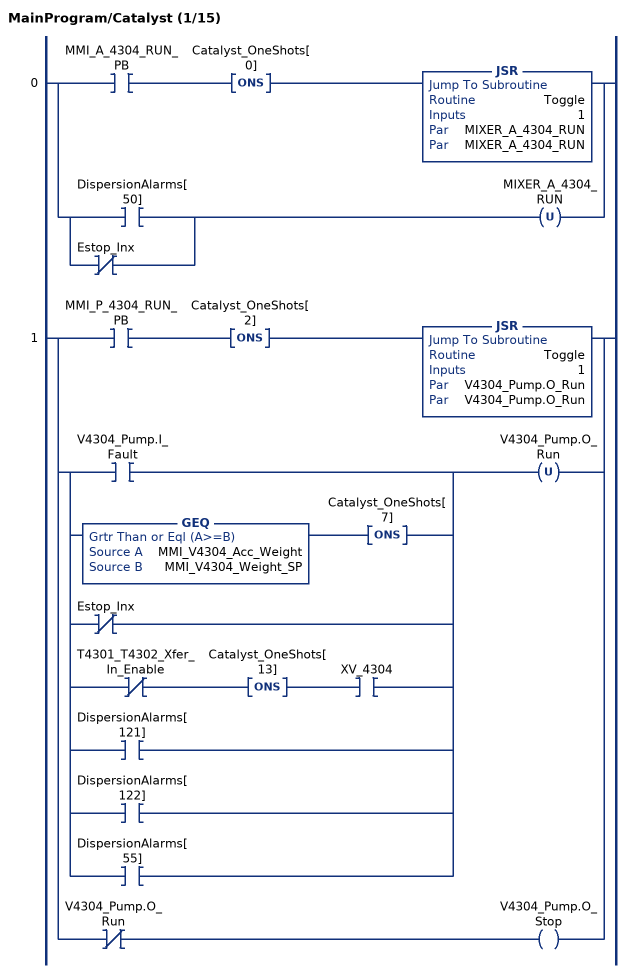
   0: [XIC(MMI_A_4304_RUN_PB) ONS(Catalyst_OneShots[0]) JSR(Toggle,1,MIXER_A_4304_RUN,MIXER_A_4304_RUN) ,[XIC(DispersionAlarms[50]) ,XIO(Estop_Inx) ] OTU(MIXER_A_4304_RUN) ];
   1: [XIC(MMI_P_4304_RUN_PB) ONS(Catalyst_OneShots[2]) JSR(Toggle,1,V4304_Pump.O_Run,V4304_Pump.O_Run) ,[XIC(V4304_Pump.I_Fault) ,GEQ(MMI_V4304_Acc_Weight,MMI_V4304_Weight_SP) ONS(Catalyst_OneShots[7]) ,XIO(Estop_Inx) ,XIO(T4301_T4302_Xfer_In_Enable) ONS(Catalyst_OneShots[13]) XIC(XV_4304) ,XIC(DispersionAlarms[121]) ,XIC(DispersionAlarms[122]) ,XIC(DispersionAlarms[55]) ] OTU(V4304_Pump.O_Run) ,XIO(V4304_Pump.O_Run) OTE(V4304_Pump.O_Stop) ];
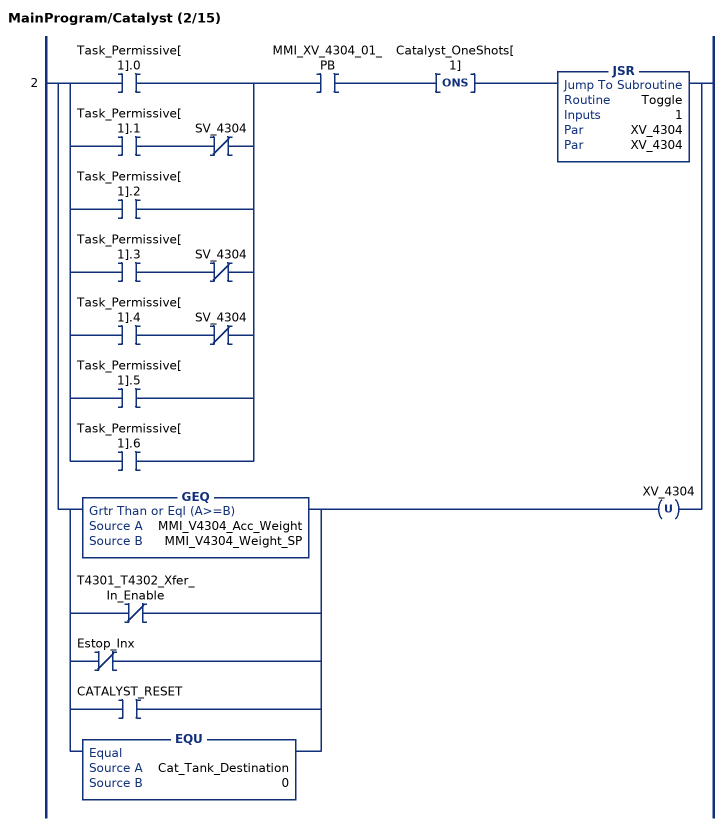
   2: [[XIC(Task_Permissive[1].0) ,XIC(Task_Permissive[1].1) XIO(SV_4304) ,XIC(Task_Permissive[1].2) ,XIC(Task_Permissive[1].3) XIO(SV_4304) ,XIC(Task_Permissive[1].4) XIO(SV_4304) ,XIC(Task_Permissive[1].5) ,XIC(Task_Permissive[1].6) ] XIC(MMI_XV_4304_01_PB) ONS(Catalyst_OneShots[1]) JSR(Toggle,1,XV_4304,XV_4304) ,[GEQ(MMI_V4304_Acc_Weight,MMI_V4304_Weight_SP) ,XIO(T4301_T4302_Xfer_In_Enable) ,XIO(Estop_Inx) ,XIC(CATALYST_RESET) ,EQU(Cat_Tank_Destination,0) ] OTU(XV_4304) ];
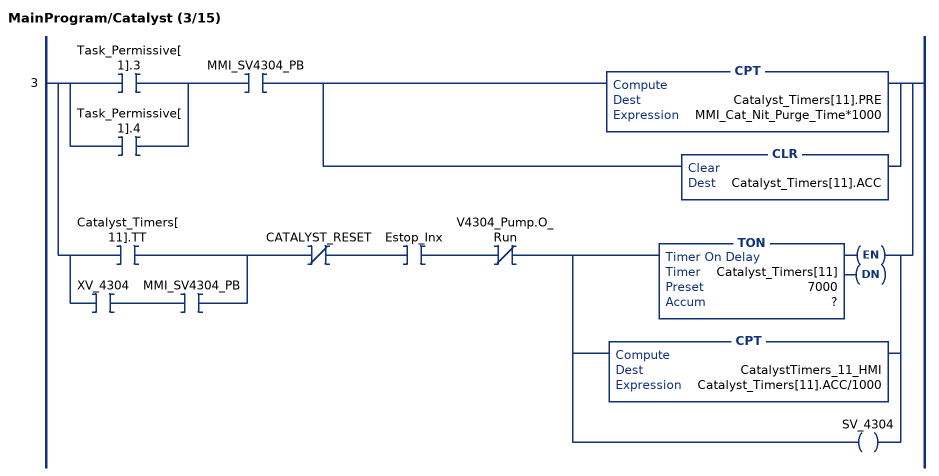
   3: [[XIC(Task_Permissive[1].3) ,XIC(Task_Permissive[1].4) ] XIC(MMI_SV4304_PB) [CPT(Catalyst_Timers[11].PRE,MMI_Cat_Nit_Purge_Time*1000) ,CLR(Catalyst_Timers[11].ACC) ] ,[XIC(Catalyst_Timers[11].TT) ,XIC(XV_4304) XIC(MMI_SV4304_PB) ] XIO(CATALYST_RESET) XIC(Estop_Inx) XIO(V4304_Pump.O_Run) [[TON(Catalyst_Timers[11],?,?) ,CPT(CatalystTimers_11_HMI,Catalyst_Timers[11].ACC/1000) ] ,OTE(SV_4304) ] ];
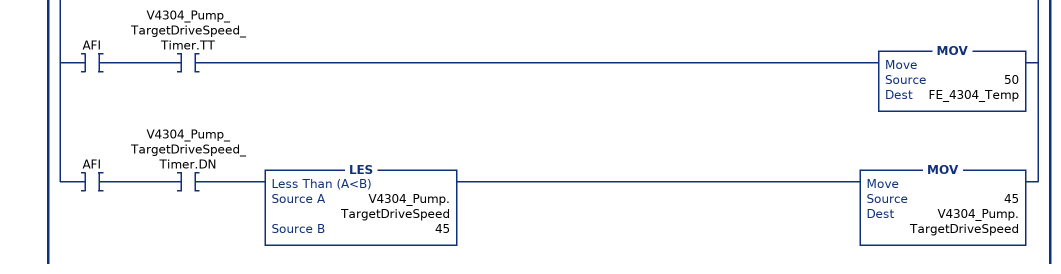
   4: [XIC(MMI_v4304_Acc_Weight_Reset) [CLR(MMI_V4304_Acc_Weight) ,CLR(MMI_V4304_Acc_Weight_Temp) ] ,LEQ(MMI_V4304_TransTime_SP,1) MOV(1,MMI_V4304_TransTime_SP) ,DIV(MMI_V4304_Weight_SP,MMI_V4304_TransTime_SP,catalyst_Target_Wgt_Lb_Min) ,XIC(cat_target_weight_bypass) GRT(catalyst_Target_Wgt_Lb_Min,catalyst_MaxFeedRate) MOV(catalyst_MaxFeedRate,catalyst_Target_Wgt_Lb_Min) ,SUB(FE_4304,catalyst_Target_Wgt_Lb_Min,FE_4304_Feed_Error) ,[XIC(XV_4304) ,XIC(Cat_Pump_manual) ] XIC(V4304_Pump.O_Run) [XIO(V4304_RampTimer.DN) TON(V4304_RampTimer,?,?) ,XIC(V4304_RampTimer.DN) [CPT(MMI_V4304_Acc_Weight,MMI_V4304_Acc_Weight+(FE_4304/(60/(V4304_RampTimer.PRE*0.001)))) ,LES(FE_4304_Feed_Error,FE_4304_Deaband_Minus) ADD(FE_4304_Temp,P4304_Rate,FE_4304_Temp) ,GRT(FE_4304_Feed_Error,FE_4304_Deaband_Plus) SUB(FE_4304_Temp,P4304_Rate,FE_4304_Temp) ] ,GRT(FE_4304_Temp,100) MOV(100,FE_4304_Temp) ,LES(FE_4304_Temp,10) MOV(10,FE_4304_Temp) ,ONS(ONS101) MOV(50,FE_4304_Temp) ,ONS(cat_start_dispencse) [CPT(calculated_percent,catalyst_Target_Wgt_Lb_Min/0.08314) ,LIM(70,calculated_percent,20) MOV(50,calculated_percent) ,MOV(calculated_percent,FE_4304_Temp) ] ,XIO(Cat_Pump_manual) MOV(FE_4304_Temp,V4304_Pump.TargetDriveSpeed) ] ,[XIO(XV_4304) ,XIO(V4304_Pump.O_Run) ] CLR(FE_4304_Temp) ,[XIO(XV_4304) ,XIC(Cat_Pump_manual) ] MOV(MMI_Cat_Recirc_Pump_Speed,V4304_Pump.TargetDriveSpeed) ,XIC(AFI) EQU(Cat_Tank_Destination,1) XIC(V4304_Pump.I_Running) XIC(XV_4304) LES(FE_4304_Temp,50) TON(V4304_Pump_TargetDriveSpeed_Timer,?,?) ,XIC(AFI) XIC(V4304_Pump_TargetDriveSpeed_Timer.TT) MOV(50,FE_4304_Temp) ,XIC(AFI) XIC(V4304_Pump_TargetDriveSpeed_Timer.DN) LES(V4304_Pump.TargetDriveSpeed,45) MOV(45,V4304_Pump.TargetDriveSpeed) ];
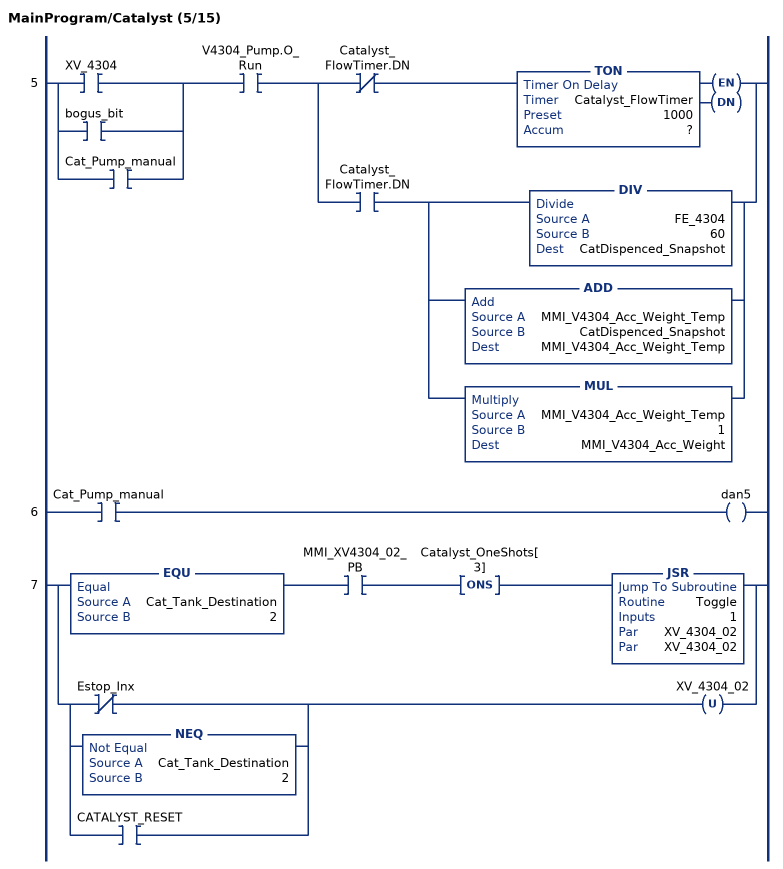
   5: [XIC(XV_4304) ,XIC(bogus_bit) ,XIC(Cat_Pump_manual) ]XIC(V4304_Pump.O_Run)[XIO(Catalyst_FlowTimer.DN) TON(Catalyst_FlowTimer,?,?) ,XIC(Catalyst_FlowTimer.DN) [DIV(FE_4304,60,CatDispenced_Snapshot) ,ADD(MMI_V4304_Acc_Weight_Temp,CatDispenced_Snapshot,MMI_V4304_Acc_Weight_Temp) ,MUL(MMI_V4304_Acc_Weight_Temp,1,MMI_V4304_Acc_Weight) ] ];
   6: XIC(Cat_Pump_manual)OTE(dan5);
   7: [EQU(Cat_Tank_Destination,2) XIC(MMI_XV4304_02_PB) ONS(Catalyst_OneShots[3]) JSR(Toggle,1,XV_4304_02,XV_4304_02) ,[XIO(Estop_Inx) ,NEQ(Cat_Tank_Destination,2) ,XIC(CATALYST_RESET) ] OTU(XV_4304_02) ];
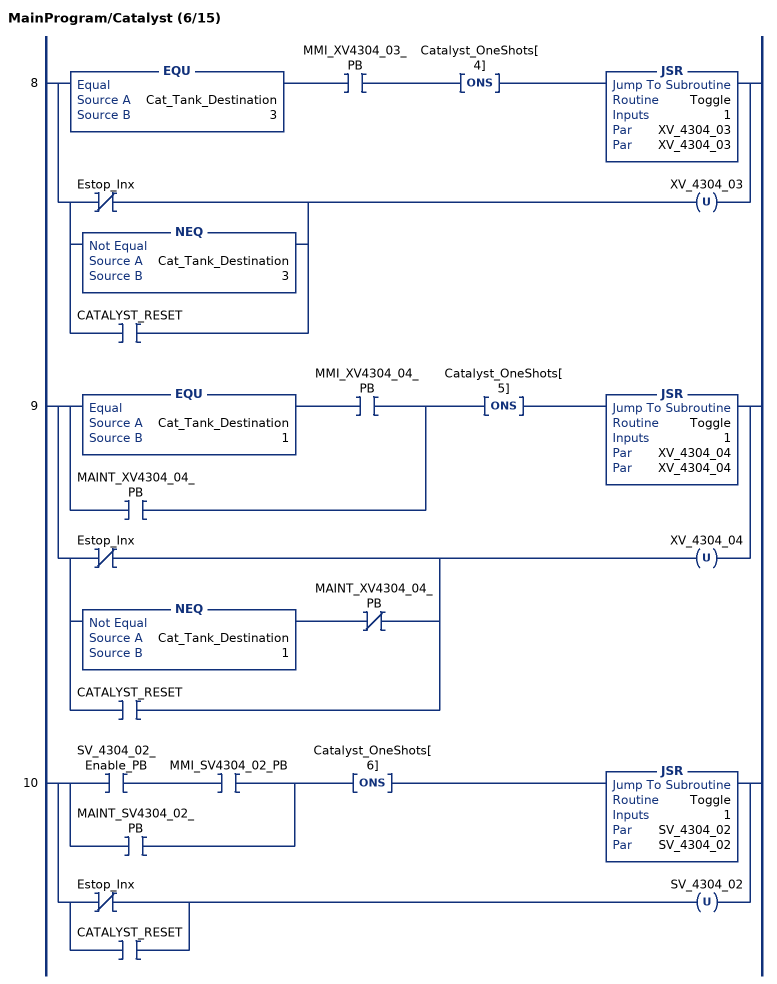
   8: [EQU(Cat_Tank_Destination,3) XIC(MMI_XV4304_03_PB) ONS(Catalyst_OneShots[4]) JSR(Toggle,1,XV_4304_03,XV_4304_03) ,[XIO(Estop_Inx) ,NEQ(Cat_Tank_Destination,3) ,XIC(CATALYST_RESET) ] OTU(XV_4304_03) ];
   9: [[EQU(Cat_Tank_Destination,1) XIC(MMI_XV4304_04_PB) ,XIC(MAINT_XV4304_04_PB) ] ONS(Catalyst_OneShots[5]) JSR(Toggle,1,XV_4304_04,XV_4304_04) ,[XIO(Estop_Inx) ,NEQ(Cat_Tank_Destination,1) XIO(MAINT_XV4304_04_PB) ,XIC(CATALYST_RESET) ] OTU(XV_4304_04) ];
   10: [[XIC(SV_4304_02_Enable_PB) XIC(MMI_SV4304_02_PB) ,XIC(MAINT_SV4304_02_PB) ] ONS(Catalyst_OneShots[6]) JSR(Toggle,1,SV_4304_02,SV_4304_02) ,[XIO(Estop_Inx) ,XIC(CATALYST_RESET) ] OTU(SV_4304_02) ];
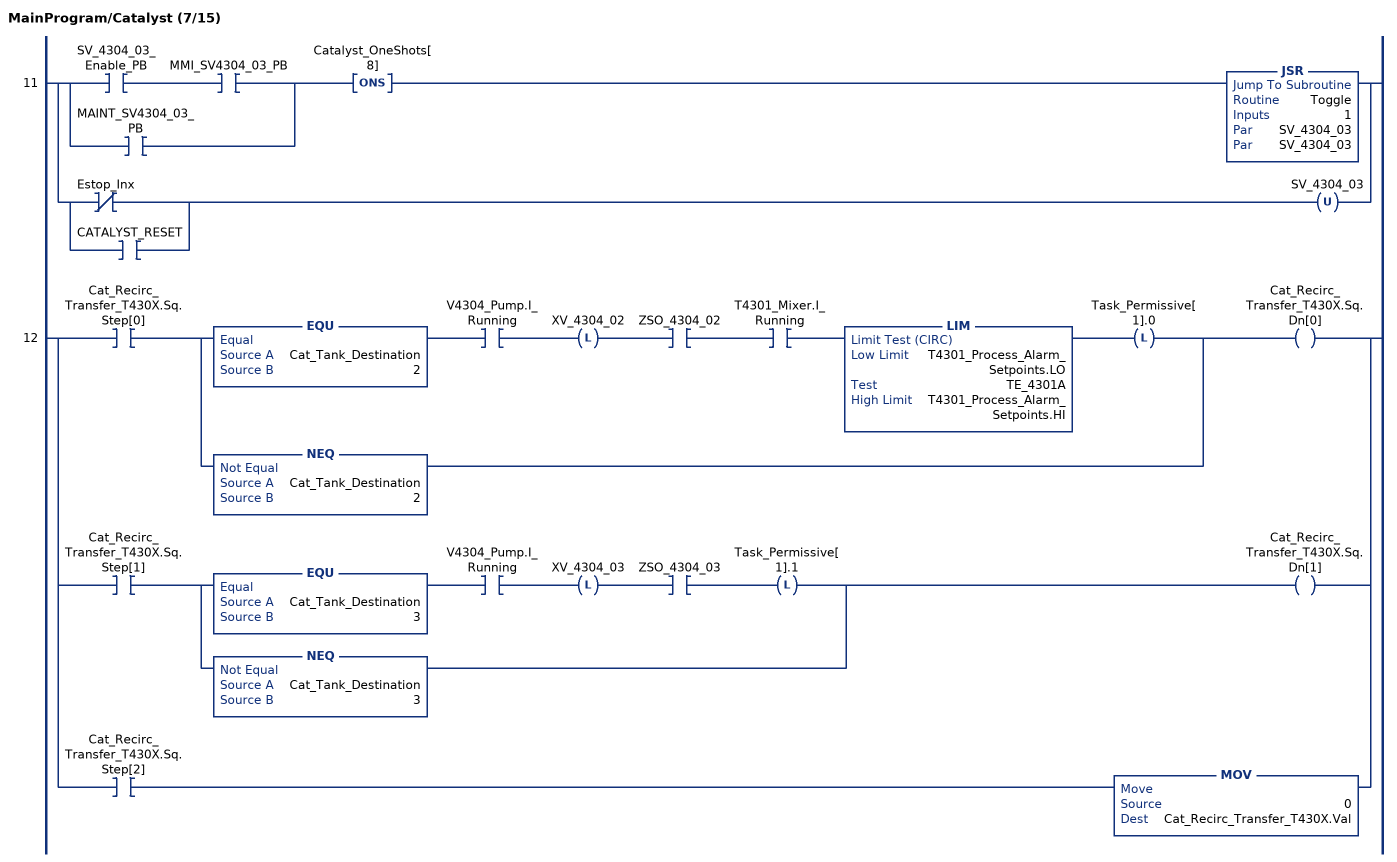
   11: [[XIC(SV_4304_03_Enable_PB) XIC(MMI_SV4304_03_PB) ,XIC(MAINT_SV4304_03_PB) ] ONS(Catalyst_OneShots[8]) JSR(Toggle,1,SV_4304_03,SV_4304_03) ,[XIO(Estop_Inx) ,XIC(CATALYST_RESET) ] OTU(SV_4304_03) ];
   12: [XIC(Cat_Recirc_Transfer_T430X.Sq.Step[0]) [EQU(Cat_Tank_Destination,2) XIC(V4304_Pump.I_Running) OTL(XV_4304_02) XIC(ZSO_4304_02) XIC(T4301_Mixer.I_Running) LIM(T4301_Process_Alarm_Setpoints.LO,TE_4301A,T4301_Process_Alarm_Setpoints.HI) OTL(Task_Permissive[1].0) ,NEQ(Cat_Tank_Destination,2) ] OTE(Cat_Recirc_Transfer_T430X.Sq.Dn[0]) ,XIC(Cat_Recirc_Transfer_T430X.Sq.Step[1]) [EQU(Cat_Tank_Destination,3) XIC(V4304_Pump.I_Running) OTL(XV_4304_03) XIC(ZSO_4304_03) OTL(Task_Permissive[1].1) ,NEQ(Cat_Tank_Destination,3) ] OTE(Cat_Recirc_Transfer_T430X.Sq.Dn[1]) ,XIC(Cat_Recirc_Transfer_T430X.Sq.Step[2]) MOV(0,Cat_Recirc_Transfer_T430X.Val) ];
